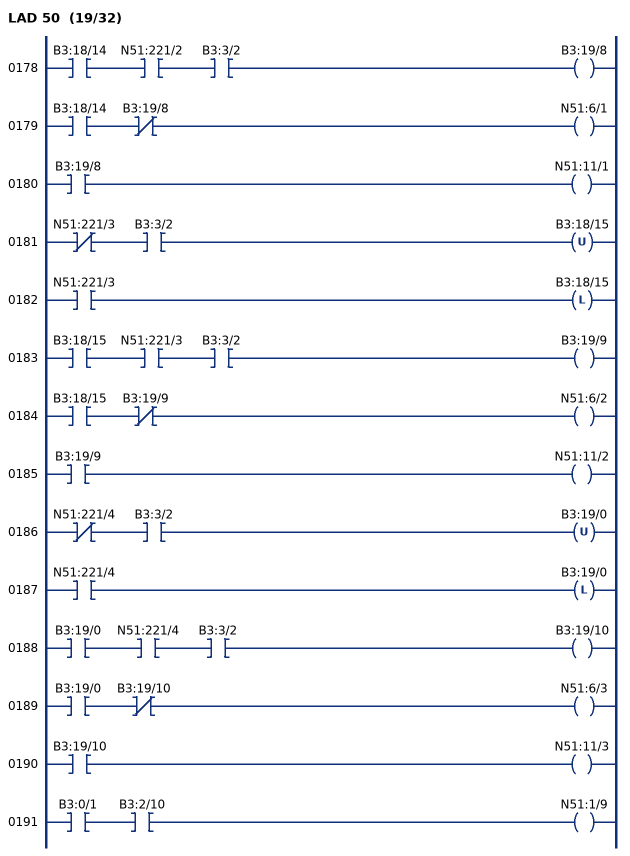
% Rung: 178 %
SOR XIC B3:18/14 XIC N51:221/2 XIC B3:3/2 OTE B3:19/8 EOR
% Rung: 179 %
SOR XIC B3:18/14 XIO B3:19/8 OTE N51:6/1 EOR
% Rung: 180 %
SOR XIC B3:19/8 OTE N51:11/1 EOR
% Rung: 181 %
SOR XIO N51:221/3 XIC B3:3/2 OTU B3:18/15 EOR
% Rung: 182 %
SOR XIC N51:221/3 OTL B3:18/15 EOR
% Rung: 183 %
SOR XIC B3:18/15 XIC N51:221/3 XIC B3:3/2 OTE B3:19/9 EOR
% Rung: 184 %
SOR XIC B3:18/15 XIO B3:19/9 OTE N51:6/2 EOR
% Rung: 185 %
SOR XIC B3:19/9 OTE N51:11/2 EOR
% Rung: 186 %
SOR XIO N51:221/4 XIC B3:3/2 OTU B3:19/0 EOR
% Rung: 187 %
SOR XIC N51:221/4 OTL B3:19/0 EOR
% Rung: 188 %
SOR XIC B3:19/0 XIC N51:221/4 XIC B3:3/2 OTE B3:19/10 EOR
% Rung: 189 %
SOR XIC B3:19/0 XIO B3:19/10 OTE N51:6/3 EOR
% Rung: 190 %
SOR XIC B3:19/10 OTE N51:11/3 EOR
% Rung: 191 %
SOR XIC B3:0/1 XIC B3:2/10 OTE N51:1/9 EOR

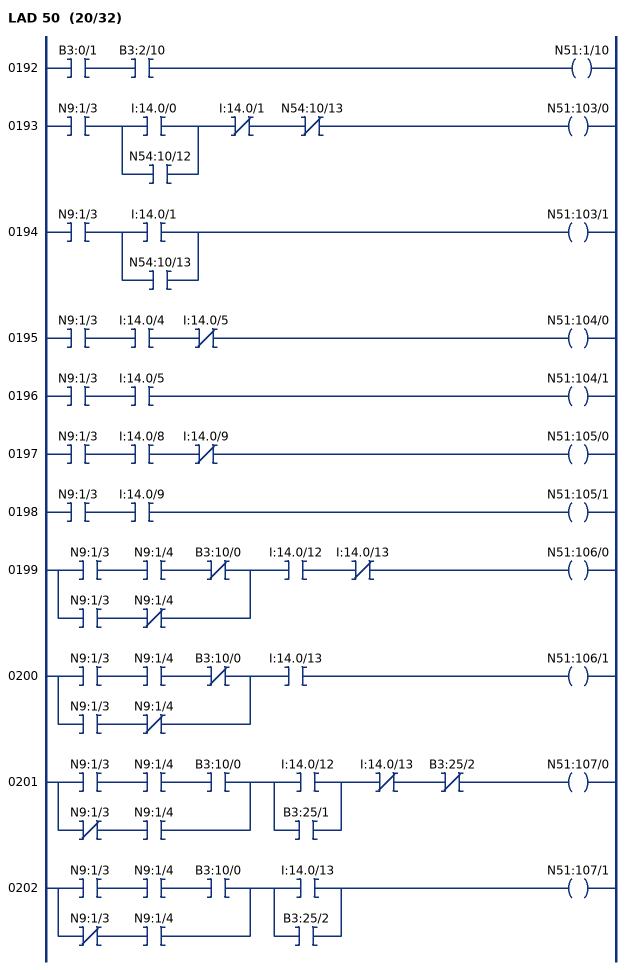
% Rung: 192 %
SOR XIC B3:0/1 XIC B3:2/10 OTE N51:1/10 EOR
% Rung: 193 %
SOR XIC N9:1/3 BST XIC I:14.0/0 NXB XIC N54:10/12 BND XIO I:14.0/1 XIO N54:10/13 OTE N51:103/0 EOR
% Rung: 194 %
SOR XIC N9:1/3 BST XIC I:14.0/1 NXB XIC N54:10/13 BND OTE N51:103/1 EOR
% Rung: 195 %
SOR XIC N9:1/3 XIC I:14.0/4 XIO I:14.0/5 OTE N51:104/0 EOR
% Rung: 196 %
SOR XIC N9:1/3 XIC I:14.0/5 OTE N51:104/1 EOR
% Rung: 197 %
SOR XIC N9:1/3 XIC I:14.0/8 XIO I:14.0/9 OTE N51:105/0 EOR
% Rung: 198 %
SOR XIC N9:1/3 XIC I:14.0/9 OTE N51:105/1 EOR
% Rung: 199 %
SOR BST XIC N9:1/3 XIC N9:1/4 XIO B3:10/0 NXB XIC N9:1/3 XIO N9:1/4 BND XIC I:14.0/12 XIO I:14.0/13 OTE N51:106/0 EOR
% Rung: 200 %
SOR BST XIC N9:1/3 XIC N9:1/4 XIO B3:10/0 NXB XIC N9:1/3 XIO N9:1/4 BND XIC I:14.0/13 OTE N51:106/1 EOR
% Rung: 201 %
SOR BST XIC N9:1/3 XIC N9:1/4 XIC B3:10/0 NXB XIO N9:1/3 XIC N9:1/4 BND BST XIC I:14.0/12 NXB XIC B3:25/1 BND XIO I:14.0/13 XIO B3:25/2 OTE N51:107/0 EOR
% Rung: 202 %
SOR BST XIC N9:1/3 XIC N9:1/4 XIC B3:10/0 NXB XIO N9:1/3 XIC N9:1/4 BND BST XIC I:14.0/13 NXB XIC B3:25/2 BND OTE N51:107/1 EOR

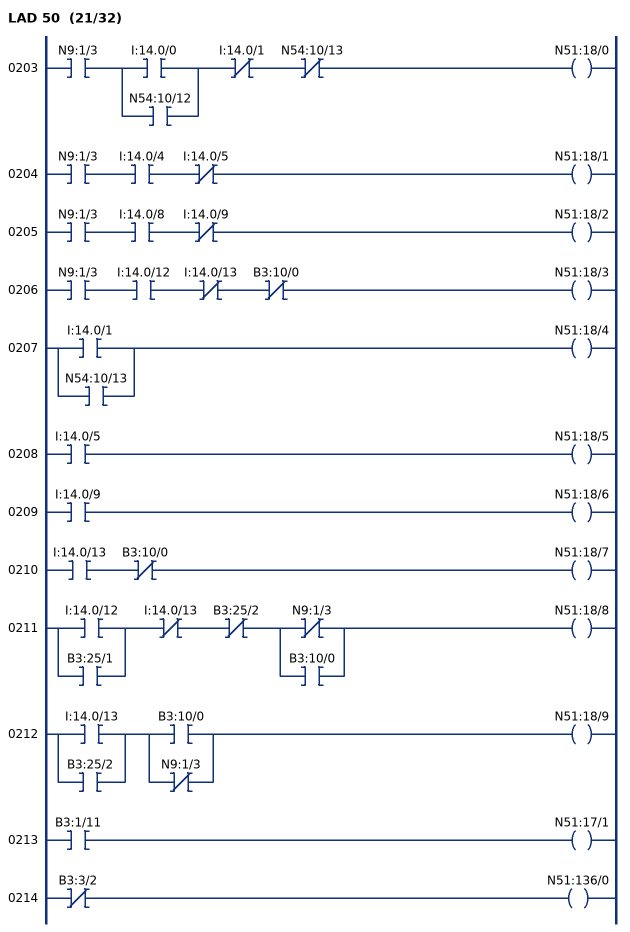
% Rung: 203 %
SOR XIC N9:1/3 BST XIC I:14.0/0 NXB XIC N54:10/12 BND XIO I:14.0/1 XIO N54:10/13 OTE N51:18/0 EOR
% Rung: 204 %
SOR XIC N9:1/3 XIC I:14.0/4 XIO I:14.0/5 OTE N51:18/1 EOR
% Rung: 205 %
SOR XIC N9:1/3 XIC I:14.0/8 XIO I:14.0/9 OTE N51:18/2 EOR
% Rung: 206 %
SOR XIC N9:1/3 XIC I:14.0/12 XIO I:14.0/13 XIO B3:10/0 OTE N51:18/3 EOR
% Rung: 207 %
SOR BST XIC I:14.0/1 NXB XIC N54:10/13 BND OTE N51:18/4 EOR
% Rung: 208 %
SOR XIC I:14.0/5 OTE N51:18/5 EOR
% Rung: 209 %
SOR XIC I:14.0/9 OTE N51:18/6 EOR
% Rung: 210 %
SOR XIC I:14.0/13 XIO B3:10/0 OTE N51:18/7 EOR
% Rung: 211 %
SOR BST XIC I:14.0/12 NXB XIC B3:25/1 BND XIO I:14.0/13 XIO B3:25/2 BST XIO N9:1/3 NXB XIC B3:10/0 BND OTE N51:18/8 EOR
% Rung: 212 %
SOR BST XIC I:14.0/13 NXB XIC B3:25/2 BND BST XIC B3:10/0 NXB XIO N9:1/3 BND OTE N51:18/9 EOR
% Rung: 213 %
SOR XIC B3:1/11 OTE N51:17/1 EOR
% Rung: 214 %
SOR XIO B3:3/2 OTE N51:136/0 EOR

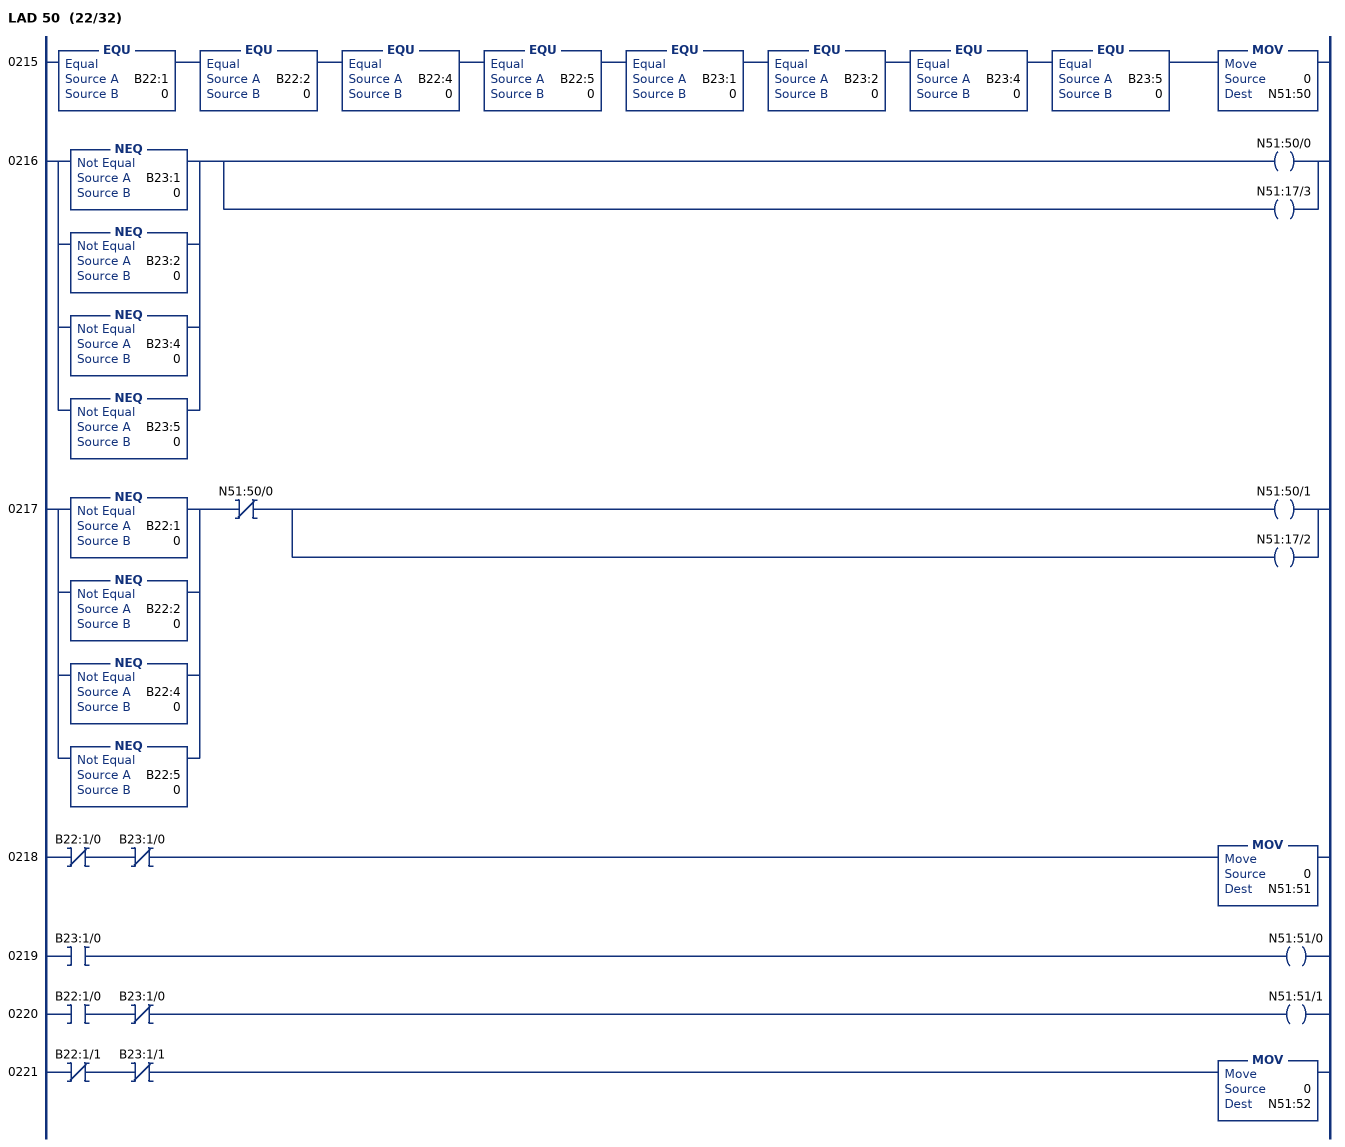
% Rung: 215 %
SOR EQU B22:1 0 EQU B22:2 0 EQU B22:4 0 EQU B22:5 0 EQU B23:1 0 EQU B23:2 0 EQU B23:4 0 EQU B23:5 0 MOV 0 N51:50 EOR
% Rung: 216 %
SOR BST NEQ B23:1 0 NXB NEQ B23:2 0 NXB NEQ B23:4 0 NXB NEQ B23:5 0 BND BST OTE N51:50/0 NXB OTE N51:17/3 BND EOR
% Rung: 217 %
SOR BST NEQ B22:1 0 NXB NEQ B22:2 0 NXB NEQ B22:4 0 NXB NEQ B22:5 0 BND XIO N51:50/0 BST OTE N51:50/1 NXB OTE N51:17/2 BND EOR
% Rung: 218 %
SOR XIO B22:1/0 XIO B23:1/0 MOV 0 N51:51 EOR
% Rung: 219 %
SOR XIC B23:1/0 OTE N51:51/0 EOR
% Rung: 220 %
SOR XIC B22:1/0 XIO B23:1/0 OTE N51:51/1 EOR
% Rung: 221 %
SOR XIO B22:1/1 XIO B23:1/1 MOV 0 N51:52 EOR

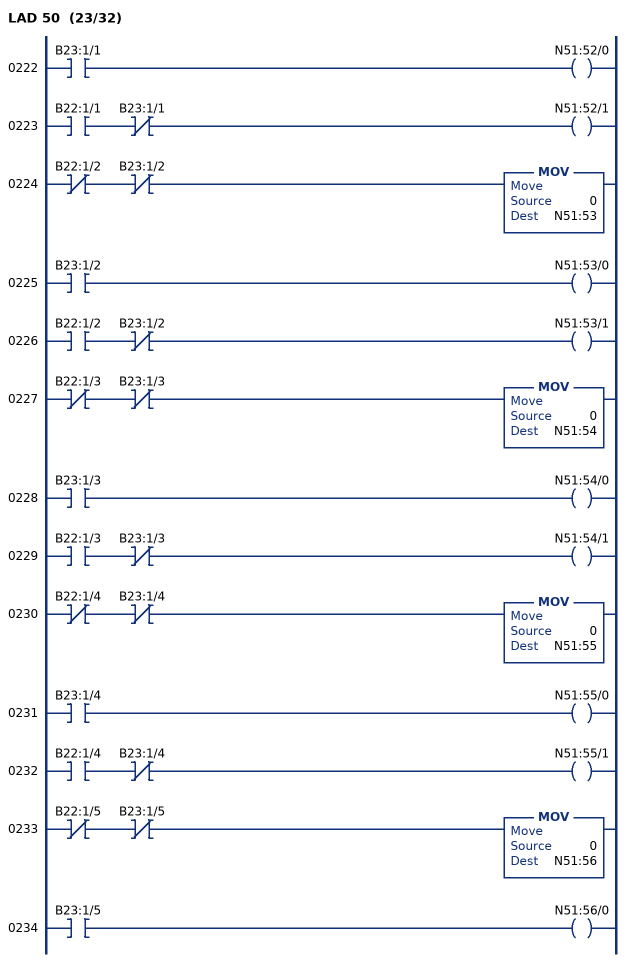
% Rung: 222 %
SOR XIC B23:1/1 OTE N51:52/0 EOR
% Rung: 223 %
SOR XIC B22:1/1 XIO B23:1/1 OTE N51:52/1 EOR
% Rung: 224 %
SOR XIO B22:1/2 XIO B23:1/2 MOV 0 N51:53 EOR
% Rung: 225 %
SOR XIC B23:1/2 OTE N51:53/0 EOR
% Rung: 226 %
SOR XIC B22:1/2 XIO B23:1/2 OTE N51:53/1 EOR
% Rung: 227 %
SOR XIO B22:1/3 XIO B23:1/3 MOV 0 N51:54 EOR
% Rung: 228 %
SOR XIC B23:1/3 OTE N51:54/0 EOR
% Rung: 229 %
SOR XIC B22:1/3 XIO B23:1/3 OTE N51:54/1 EOR
% Rung: 230 %
SOR XIO B22:1/4 XIO B23:1/4 MOV 0 N51:55 EOR
% Rung: 231 %
SOR XIC B23:1/4 OTE N51:55/0 EOR
% Rung: 232 %
SOR XIC B22:1/4 XIO B23:1/4 OTE N51:55/1 EOR
% Rung: 233 %
SOR XIO B22:1/5 XIO B23:1/5 MOV 0 N51:56 EOR
% Rung: 234 %
SOR XIC B23:1/5 OTE N51:56/0 EOR

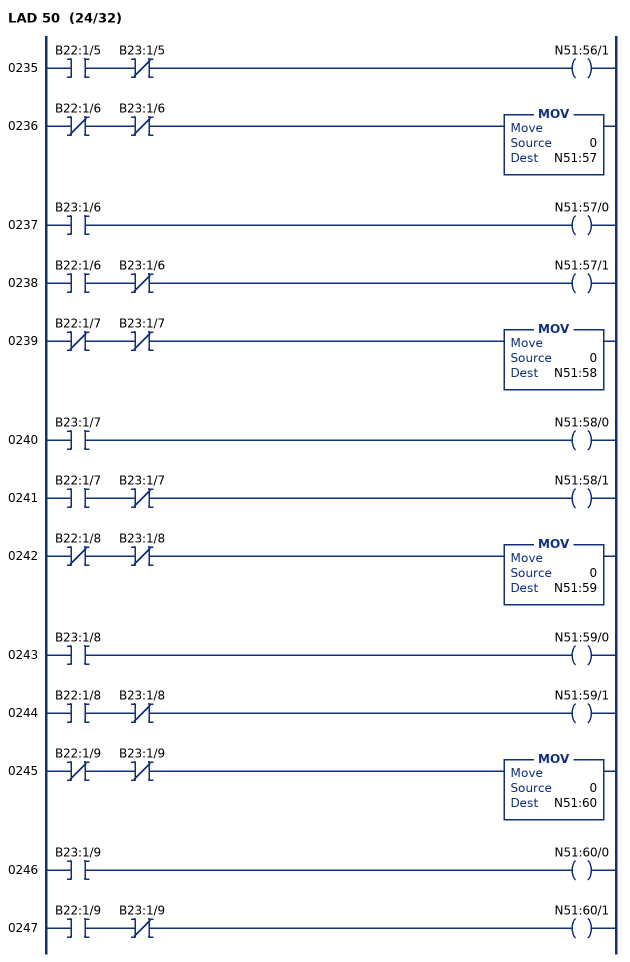
% Rung: 235 %
SOR XIC B22:1/5 XIO B23:1/5 OTE N51:56/1 EOR
% Rung: 236 %
SOR XIO B22:1/6 XIO B23:1/6 MOV 0 N51:57 EOR
% Rung: 237 %
SOR XIC B23:1/6 OTE N51:57/0 EOR
% Rung: 238 %
SOR XIC B22:1/6 XIO B23:1/6 OTE N51:57/1 EOR
% Rung: 239 %
SOR XIO B22:1/7 XIO B23:1/7 MOV 0 N51:58 EOR
% Rung: 240 %
SOR XIC B23:1/7 OTE N51:58/0 EOR
% Rung: 241 %
SOR XIC B22:1/7 XIO B23:1/7 OTE N51:58/1 EOR
% Rung: 242 %
SOR XIO B22:1/8 XIO B23:1/8 MOV 0 N51:59 EOR
% Rung: 243 %
SOR XIC B23:1/8 OTE N51:59/0 EOR
% Rung: 244 %
SOR XIC B22:1/8 XIO B23:1/8 OTE N51:59/1 EOR
% Rung: 245 %
SOR XIO B22:1/9 XIO B23:1/9 MOV 0 N51:60 EOR
% Rung: 246 %
SOR XIC B23:1/9 OTE N51:60/0 EOR
% Rung: 247 %
SOR XIC B22:1/9 XIO B23:1/9 OTE N51:60/1 EOR

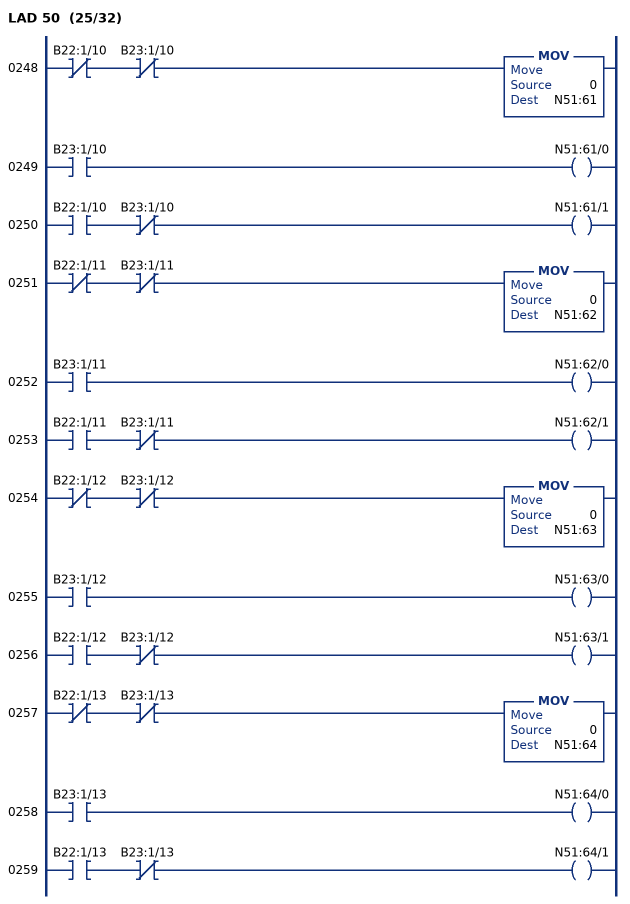
% Rung: 248 %
SOR XIO B22:1/10 XIO B23:1/10 MOV 0 N51:61 EOR
% Rung: 249 %
SOR XIC B23:1/10 OTE N51:61/0 EOR
% Rung: 250 %
SOR XIC B22:1/10 XIO B23:1/10 OTE N51:61/1 EOR
% Rung: 251 %
SOR XIO B22:1/11 XIO B23:1/11 MOV 0 N51:62 EOR
% Rung: 252 %
SOR XIC B23:1/11 OTE N51:62/0 EOR
% Rung: 253 %
SOR XIC B22:1/11 XIO B23:1/11 OTE N51:62/1 EOR
% Rung: 254 %
SOR XIO B22:1/12 XIO B23:1/12 MOV 0 N51:63 EOR
% Rung: 255 %
SOR XIC B23:1/12 OTE N51:63/0 EOR
% Rung: 256 %
SOR XIC B22:1/12 XIO B23:1/12 OTE N51:63/1 EOR
% Rung: 257 %
SOR XIO B22:1/13 XIO B23:1/13 MOV 0 N51:64 EOR
% Rung: 258 %
SOR XIC B23:1/13 OTE N51:64/0 EOR
% Rung: 259 %
SOR XIC B22:1/13 XIO B23:1/13 OTE N51:64/1 EOR

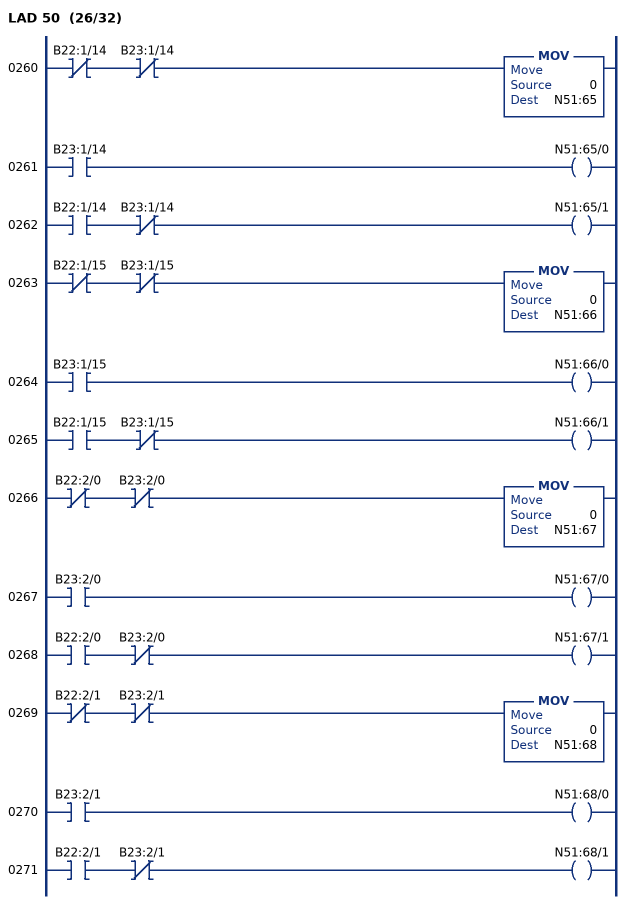
% Rung: 260 %
SOR XIO B22:1/14 XIO B23:1/14 MOV 0 N51:65 EOR
% Rung: 261 %
SOR XIC B23:1/14 OTE N51:65/0 EOR
% Rung: 262 %
SOR XIC B22:1/14 XIO B23:1/14 OTE N51:65/1 EOR
% Rung: 263 %
SOR XIO B22:1/15 XIO B23:1/15 MOV 0 N51:66 EOR
% Rung: 264 %
SOR XIC B23:1/15 OTE N51:66/0 EOR
% Rung: 265 %
SOR XIC B22:1/15 XIO B23:1/15 OTE N51:66/1 EOR
% Rung: 266 %
SOR XIO B22:2/0 XIO B23:2/0 MOV 0 N51:67 EOR
% Rung: 267 %
SOR XIC B23:2/0 OTE N51:67/0 EOR
% Rung: 268 %
SOR XIC B22:2/0 XIO B23:2/0 OTE N51:67/1 EOR
% Rung: 269 %
SOR XIO B22:2/1 XIO B23:2/1 MOV 0 N51:68 EOR
% Rung: 270 %
SOR XIC B23:2/1 OTE N51:68/0 EOR
% Rung: 271 %
SOR XIC B22:2/1 XIO B23:2/1 OTE N51:68/1 EOR

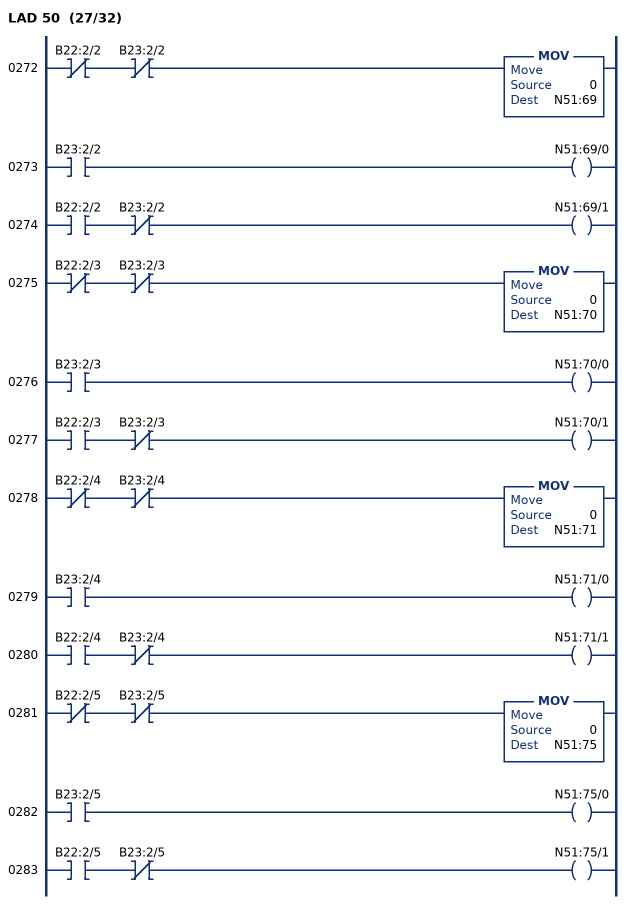
% Rung: 272 %
SOR XIO B22:2/2 XIO B23:2/2 MOV 0 N51:69 EOR
% Rung: 273 %
SOR XIC B23:2/2 OTE N51:69/0 EOR
% Rung: 274 %
SOR XIC B22:2/2 XIO B23:2/2 OTE N51:69/1 EOR
% Rung: 275 %
SOR XIO B22:2/3 XIO B23:2/3 MOV 0 N51:70 EOR
% Rung: 276 %
SOR XIC B23:2/3 OTE N51:70/0 EOR
% Rung: 277 %
SOR XIC B22:2/3 XIO B23:2/3 OTE N51:70/1 EOR
% Rung: 278 %
SOR XIO B22:2/4 XIO B23:2/4 MOV 0 N51:71 EOR
% Rung: 279 %
SOR XIC B23:2/4 OTE N51:71/0 EOR
% Rung: 280 %
SOR XIC B22:2/4 XIO B23:2/4 OTE N51:71/1 EOR
% Rung: 281 %
SOR XIO B22:2/5 XIO B23:2/5 MOV 0 N51:75 EOR
% Rung: 282 %
SOR XIC B23:2/5 OTE N51:75/0 EOR
% Rung: 283 %
SOR XIC B22:2/5 XIO B23:2/5 OTE N51:75/1 EOR

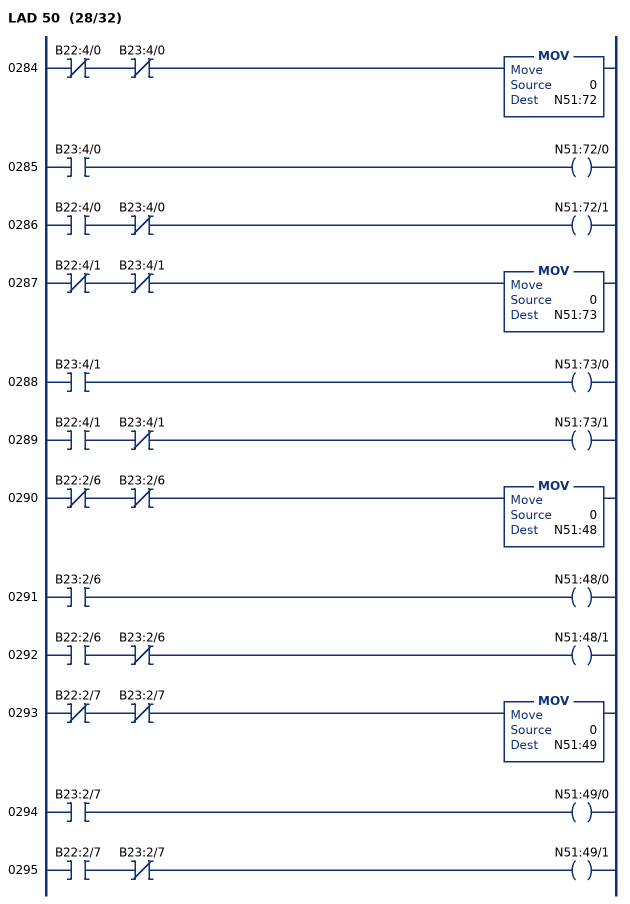
% Rung: 284 %
SOR XIO B22:4/0 XIO B23:4/0 MOV 0 N51:72 EOR
% Rung: 285 %
SOR XIC B23:4/0 OTE N51:72/0 EOR
% Rung: 286 %
SOR XIC B22:4/0 XIO B23:4/0 OTE N51:72/1 EOR
% Rung: 287 %
SOR XIO B22:4/1 XIO B23:4/1 MOV 0 N51:73 EOR
% Rung: 288 %
SOR XIC B23:4/1 OTE N51:73/0 EOR
% Rung: 289 %
SOR XIC B22:4/1 XIO B23:4/1 OTE N51:73/1 EOR
% Rung: 290 %
SOR XIO B22:2/6 XIO B23:2/6 MOV 0 N51:48 EOR
% Rung: 291 %
SOR XIC B23:2/6 OTE N51:48/0 EOR
% Rung: 292 %
SOR XIC B22:2/6 XIO B23:2/6 OTE N51:48/1 EOR
% Rung: 293 %
SOR XIO B22:2/7 XIO B23:2/7 MOV 0 N51:49 EOR
% Rung: 294 %
SOR XIC B23:2/7 OTE N51:49/0 EOR
% Rung: 295 %
SOR XIC B22:2/7 XIO B23:2/7 OTE N51:49/1 EOR

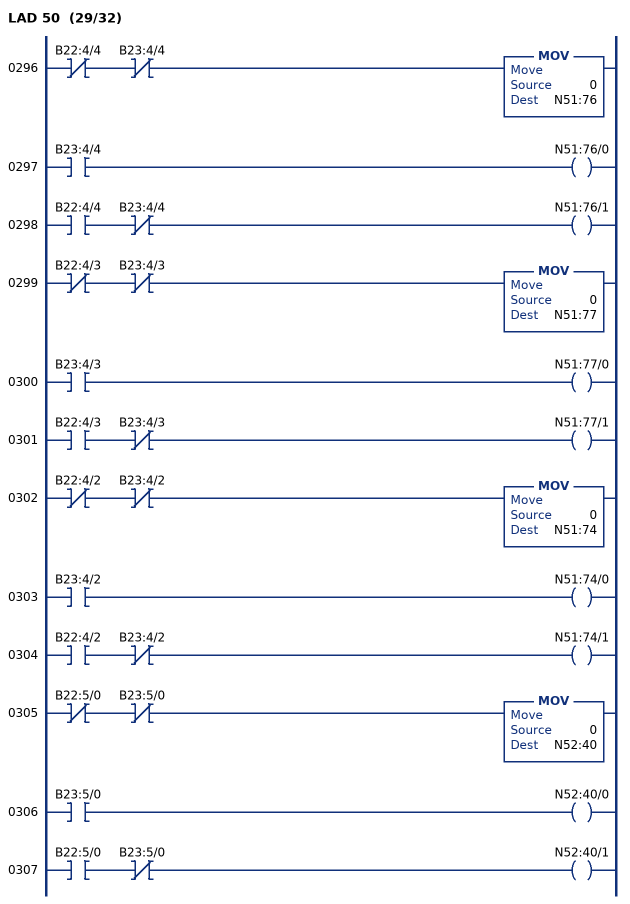
% Rung: 296 %
SOR XIO B22:4/4 XIO B23:4/4 MOV 0 N51:76 EOR
% Rung: 297 %
SOR XIC B23:4/4 OTE N51:76/0 EOR
% Rung: 298 %
SOR XIC B22:4/4 XIO B23:4/4 OTE N51:76/1 EOR
% Rung: 299 %
SOR XIO B22:4/3 XIO B23:4/3 MOV 0 N51:77 EOR
% Rung: 300 %
SOR XIC B23:4/3 OTE N51:77/0 EOR
% Rung: 301 %
SOR XIC B22:4/3 XIO B23:4/3 OTE N51:77/1 EOR
% Rung: 302 %
SOR XIO B22:4/2 XIO B23:4/2 MOV 0 N51:74 EOR
% Rung: 303 %
SOR XIC B23:4/2 OTE N51:74/0 EOR
% Rung: 304 %
SOR XIC B22:4/2 XIO B23:4/2 OTE N51:74/1 EOR
% Rung: 305 %
SOR XIO B22:5/0 XIO B23:5/0 MOV 0 N52:40 EOR
% Rung: 306 %
SOR XIC B23:5/0 OTE N52:40/0 EOR
% Rung: 307 %
SOR XIC B22:5/0 XIO B23:5/0 OTE N52:40/1 EOR

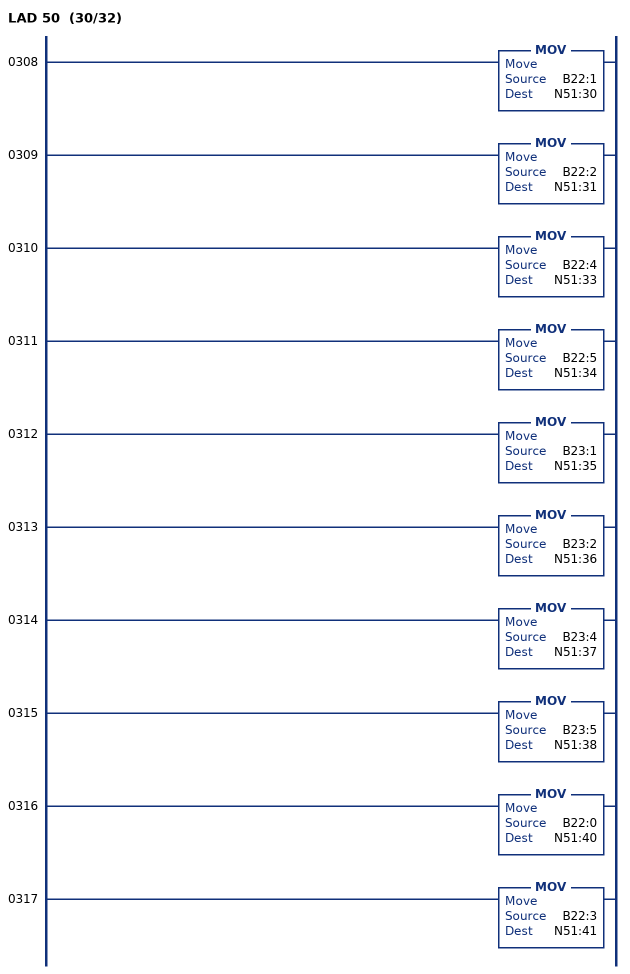
% Rung: 308 %
SOR MOV B22:1 N51:30 EOR
% Rung: 309 %
SOR MOV B22:2 N51:31 EOR
% Rung: 310 %
SOR MOV B22:4 N51:33 EOR
% Rung: 311 %
SOR MOV B22:5 N51:34 EOR
% Rung: 312 %
SOR MOV B23:1 N51:35 EOR
% Rung: 313 %
SOR MOV B23:2 N51:36 EOR
% Rung: 314 %
SOR MOV B23:4 N51:37 EOR
% Rung: 315 %
SOR MOV B23:5 N51:38 EOR
% Rung: 316 %
SOR MOV B22:0 N51:40 EOR
% Rung: 317 %
SOR MOV B22:3 N51:41 EOR

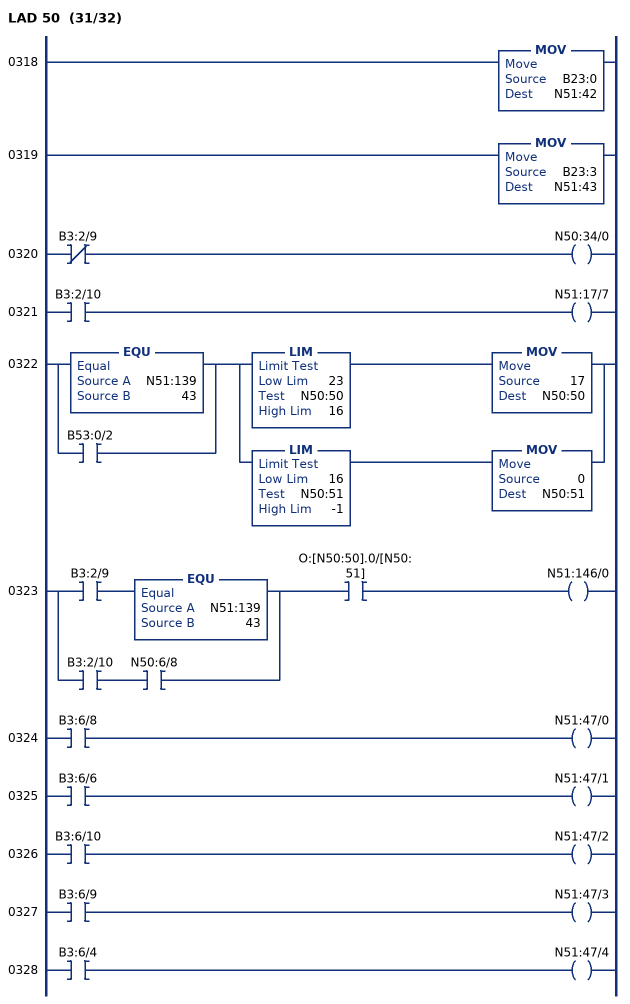
% Rung: 318 %
SOR MOV B23:0 N51:42 EOR
% Rung: 319 %
SOR MOV B23:3 N51:43 EOR
% Rung: 320 %
SOR XIO B3:2/9 OTE N50:34/0 EOR
% Rung: 321 %
SOR XIC B3:2/10 OTE N51:17/7 EOR
% Rung: 322 %
SOR BST EQU N51:139 43 NXB XIC B53:0/2 BND BST LIM 23 N50:50 16 MOV 17 N50:50 NXB LIM 16 N50:51 -1 MOV 0 N50:51 BND EOR
% Rung: 323 %
SOR BST XIC B3:2/9 EQU N51:139 43 NXB XIC B3:2/10 XIC N50:6/8 BND XIC O:[N50:50].0/[N50:51] OTE N51:146/0 EOR
% Rung: 324 %
SOR XIC B3:6/8 OTE N51:47/0 EOR
% Rung: 325 %
SOR XIC B3:6/6 OTE N51:47/1 EOR
% Rung: 326 %
SOR XIC B3:6/10 OTE N51:47/2 EOR
% Rung: 327 %
SOR XIC B3:6/9 OTE N51:47/3 EOR
% Rung: 328 %
SOR XIC B3:6/4 OTE N51:47/4 EOR

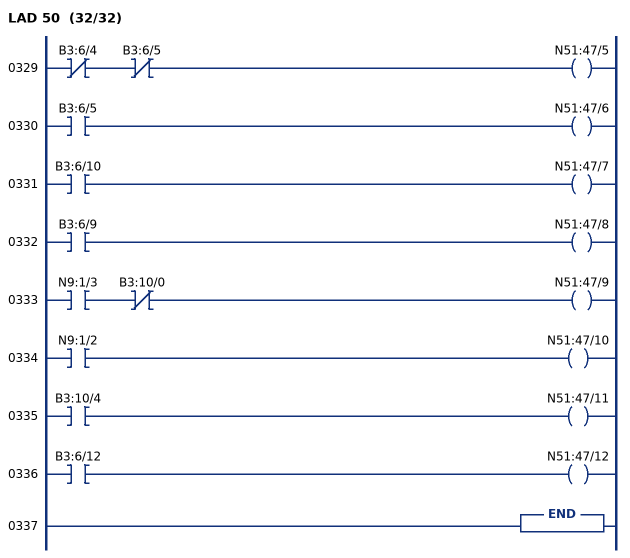
% Rung: 329 %
SOR XIO B3:6/4 XIO B3:6/5 OTE N51:47/5 EOR
% Rung: 330 %
SOR XIC B3:6/5 OTE N51:47/6 EOR
% Rung: 331 %
SOR XIC B3:6/10 OTE N51:47/7 EOR
% Rung: 332 %
SOR XIC B3:6/9 OTE N51:47/8 EOR
% Rung: 333 %
SOR XIC N9:1/3 XIO B3:10/0 OTE N51:47/9 EOR
% Rung: 334 %
SOR XIC N9:1/2 OTE N51:47/10 EOR
% Rung: 335 %
SOR XIC B3:10/4 OTE N51:47/11 EOR
% Rung: 336 %
SOR XIC B3:6/12 OTE N51:47/12 EOR
% Rung: 337 %
SOR END EOR

LADDER 51
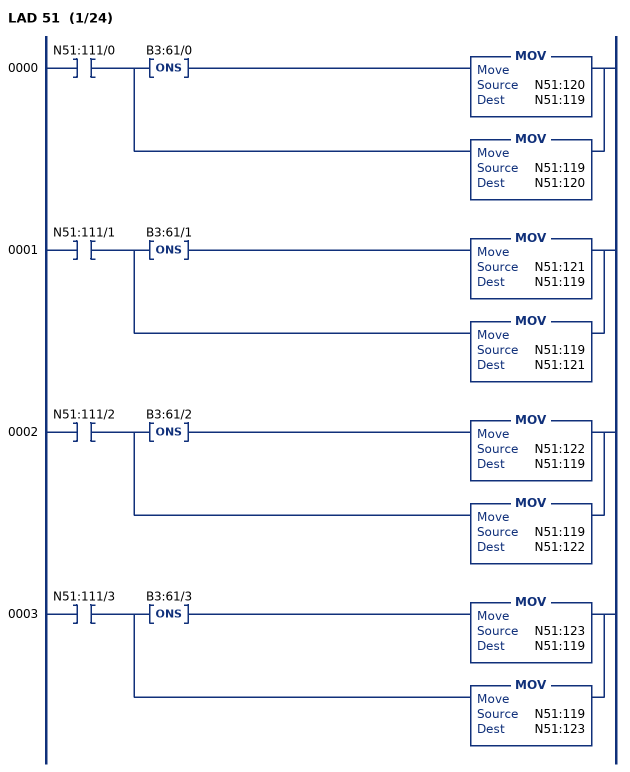
% Rung: 0 %
SOR XIC N51:111/0 BST OSR B3:61/0 MOV N51:120 N51:119 NXB MOV N51:119 N51:120 BND EOR
% Rung: 1 %
SOR XIC N51:111/1 BST OSR B3:61/1 MOV N51:121 N51:119 NXB MOV N51:119 N51:121 BND EOR
% Rung: 2 %
SOR XIC N51:111/2 BST OSR B3:61/2 MOV N51:122 N51:119 NXB MOV N51:119 N51:122 BND EOR
% Rung: 3 %
SOR XIC N51:111/3 BST OSR B3:61/3 MOV N51:123 N51:119 NXB MOV N51:119 N51:123 BND EOR

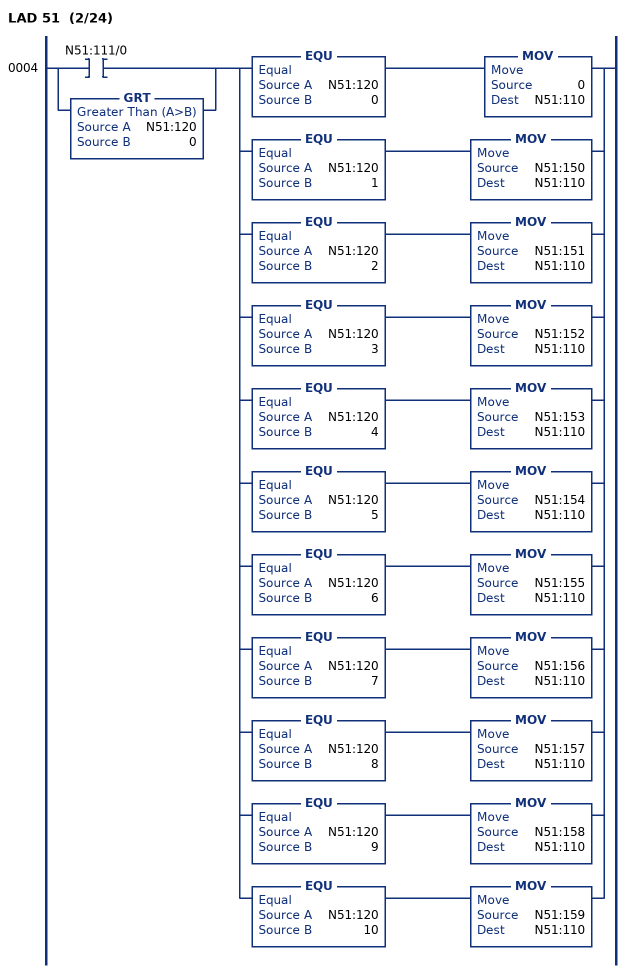
% Rung: 4 %
SOR BST XIC N51:111/0 NXB GRT N51:120 0 BND BST EQU N51:120 0 MOV 0 N51:110 NXB EQU N51:120 1 MOV N51:150 N51:110 NXB EQU N51:120 2 MOV N51:151 N51:110 NXB EQU N51:120 3 MOV N51:152 N51:110 NXB EQU N51:120 4 MOV N51:153 N51:110 NXB EQU N51:120 5 MOV N51:154 N51:110 NXB EQU N51:120 6 MOV N51:155 N51:110 NXB EQU N51:120 7 MOV N51:156 N51:110 NXB EQU N51:120 8 MOV N51:157 N51:110 NXB EQU N51:120 9 MOV N51:158 N51:110 NXB EQU N51:120 10 MOV N51:159 N51:110 BND EOR

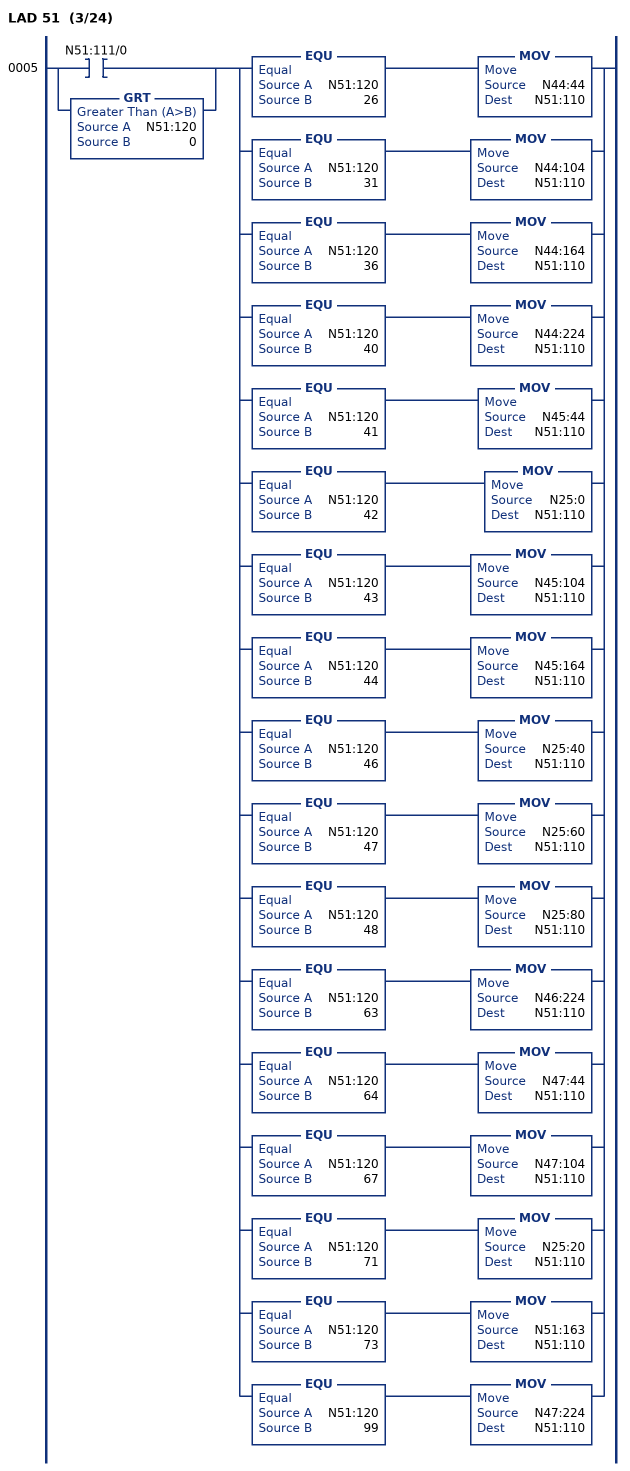
% Rung: 5 %
SOR BST XIC N51:111/0 NXB GRT N51:120 0 BND BST EQU N51:120 26 MOV N44:44 N51:110 NXB EQU N51:120 31 MOV N44:104 N51:110 NXB EQU N51:120 36 MOV N44:164 N51:110 NXB EQU N51:120 40 MOV N44:224 N51:110 NXB EQU N51:120 41 MOV N45:44 N51:110 NXB EQU N51:120 42 MOV N25:0 N51:110 NXB EQU N51:120 43 MOV N45:104 N51:110 NXB EQU N51:120 44 MOV N45:164 N51:110 NXB EQU N51:120 46 MOV N25:40 N51:110 NXB EQU N51:120 47 MOV N25:60 N51:110 NXB EQU N51:120 48 MOV N25:80 N51:110 NXB EQU N51:120 63 MOV N46:224 N51:110 NXB EQU N51:120 64 MOV N47:44 N51:110 NXB EQU N51:120 67 MOV N47:104 N51:110 NXB EQU N51:120 71 MOV N25:20 N51:110 NXB EQU N51:120 73 MOV N51:163 N51:110 NXB EQU N51:120 99 MOV N47:224 N51:110 BND EOR

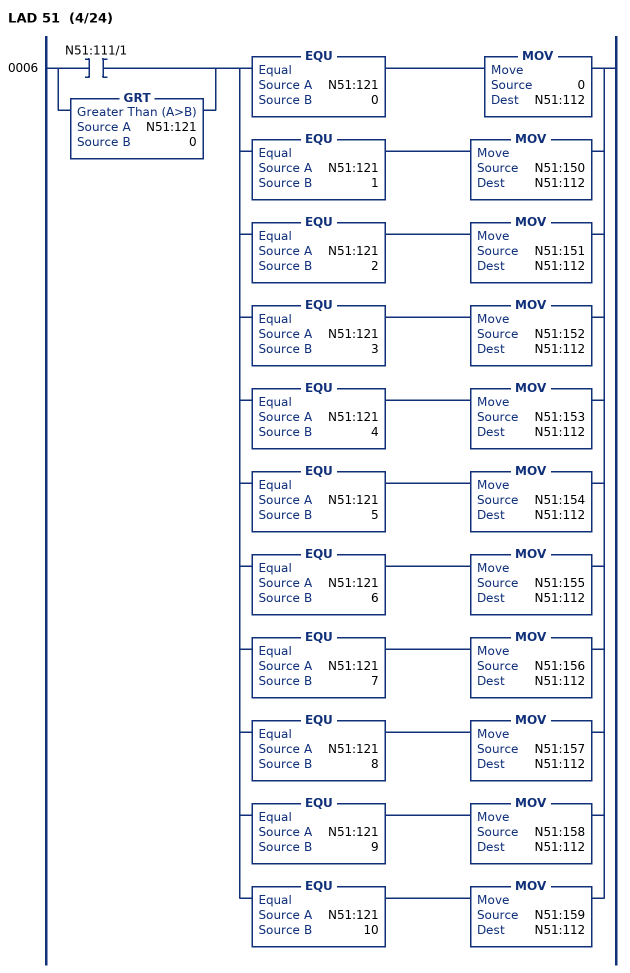
% Rung: 6 %
SOR BST XIC N51:111/1 NXB GRT N51:121 0 BND BST EQU N51:121 0 MOV 0 N51:112 NXB EQU N51:121 1 MOV N51:150 N51:112 NXB EQU N51:121 2 MOV N51:151 N51:112 NXB EQU N51:121 3 MOV N51:152 N51:112 NXB EQU N51:121 4 MOV N51:153 N51:112 NXB EQU N51:121 5 MOV N51:154 N51:112 NXB EQU N51:121 6 MOV N51:155 N51:112 NXB EQU N51:121 7 MOV N51:156 N51:112 NXB EQU N51:121 8 MOV N51:157 N51:112 NXB EQU N51:121 9 MOV N51:158 N51:112 NXB EQU N51:121 10 MOV N51:159 N51:112 BND EOR

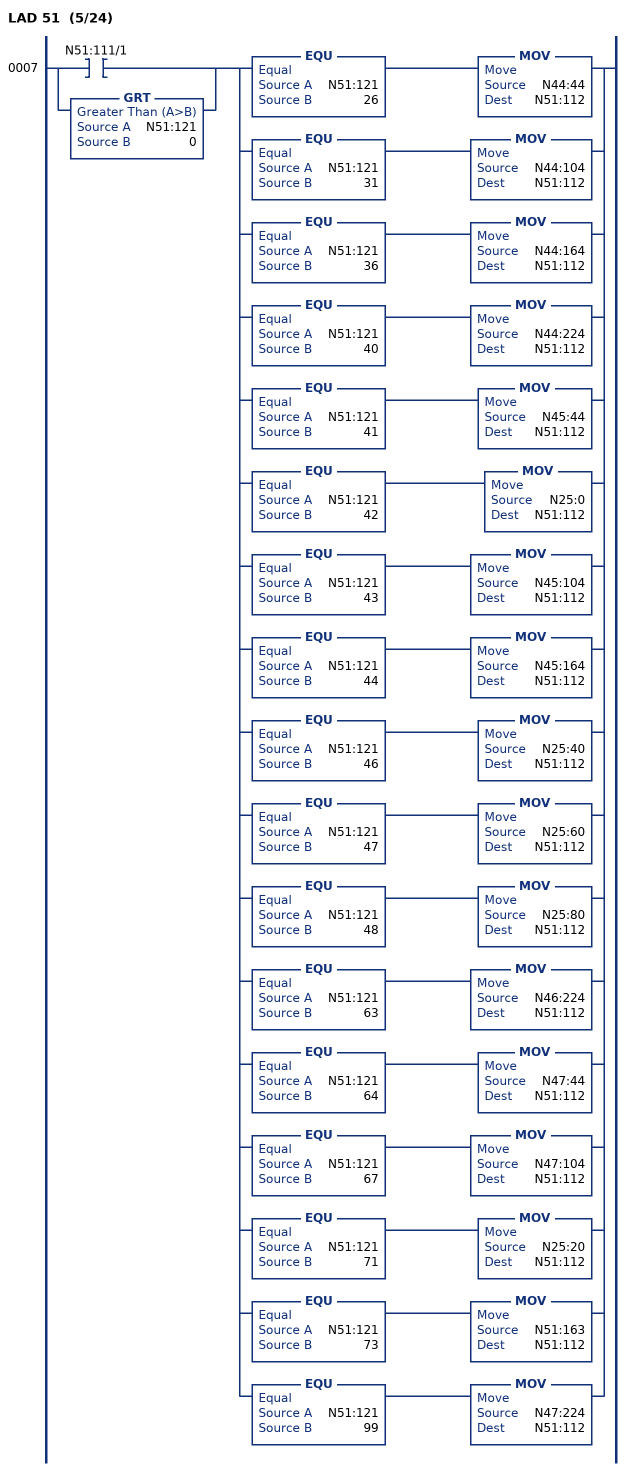
% Rung: 7 %
SOR BST XIC N51:111/1 NXB GRT N51:121 0 BND BST EQU N51:121 26 MOV N44:44 N51:112 NXB EQU N51:121 31 MOV N44:104 N51:112 NXB EQU N51:121 36 MOV N44:164 N51:112 NXB EQU N51:121 40 MOV N44:224 N51:112 NXB EQU N51:121 41 MOV N45:44 N51:112 NXB EQU N51:121 42 MOV N25:0 N51:112 NXB EQU N51:121 43 MOV N45:104 N51:112 NXB EQU N51:121 44 MOV N45:164 N51:112 NXB EQU N51:121 46 MOV N25:40 N51:112 NXB EQU N51:121 47 MOV N25:60 N51:112 NXB EQU N51:121 48 MOV N25:80 N51:112 NXB EQU N51:121 63 MOV N46:224 N51:112 NXB EQU N51:121 64 MOV N47:44 N51:112 NXB EQU N51:121 67 MOV N47:104 N51:112 NXB EQU N51:121 71 MOV N25:20 N51:112 NXB EQU N51:121 73 MOV N51:163 N51:112 NXB EQU N51:121 99 MOV N47:224 N51:112 BND EOR

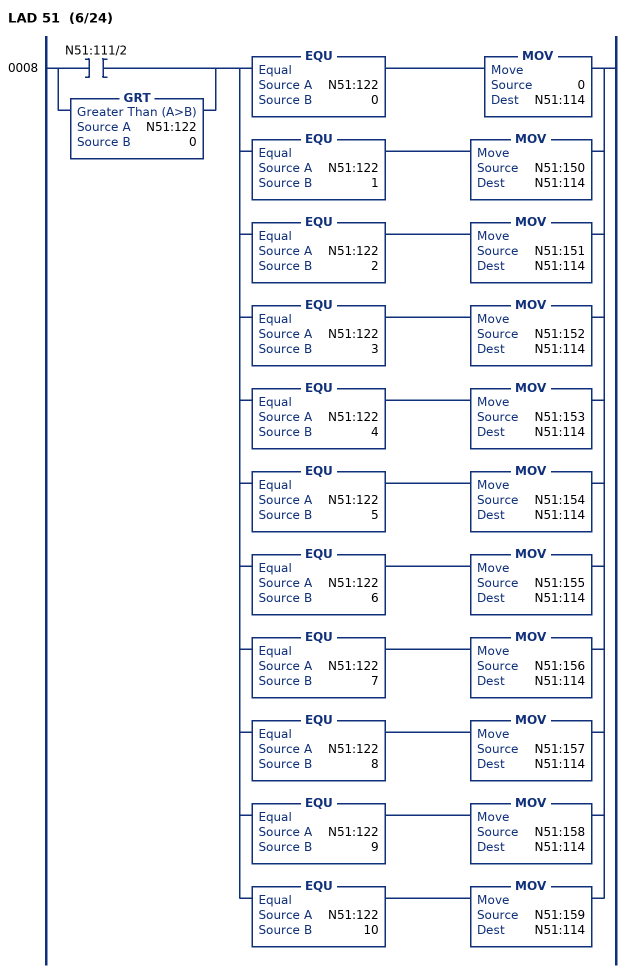
% Rung: 8 %
SOR BST XIC N51:111/2 NXB GRT N51:122 0 BND BST EQU N51:122 0 MOV 0 N51:114 NXB EQU N51:122 1 MOV N51:150 N51:114 NXB EQU N51:122 2 MOV N51:151 N51:114 NXB EQU N51:122 3 MOV N51:152 N51:114 NXB EQU N51:122 4 MOV N51:153 N51:114 NXB EQU N51:122 5 MOV N51:154 N51:114 NXB EQU N51:122 6 MOV N51:155 N51:114 NXB EQU N51:122 7 MOV N51:156 N51:114 NXB EQU N51:122 8 MOV N51:157 N51:114 NXB EQU N51:122 9 MOV N51:158 N51:114 NXB EQU N51:122 10 MOV N51:159 N51:114 BND EOR

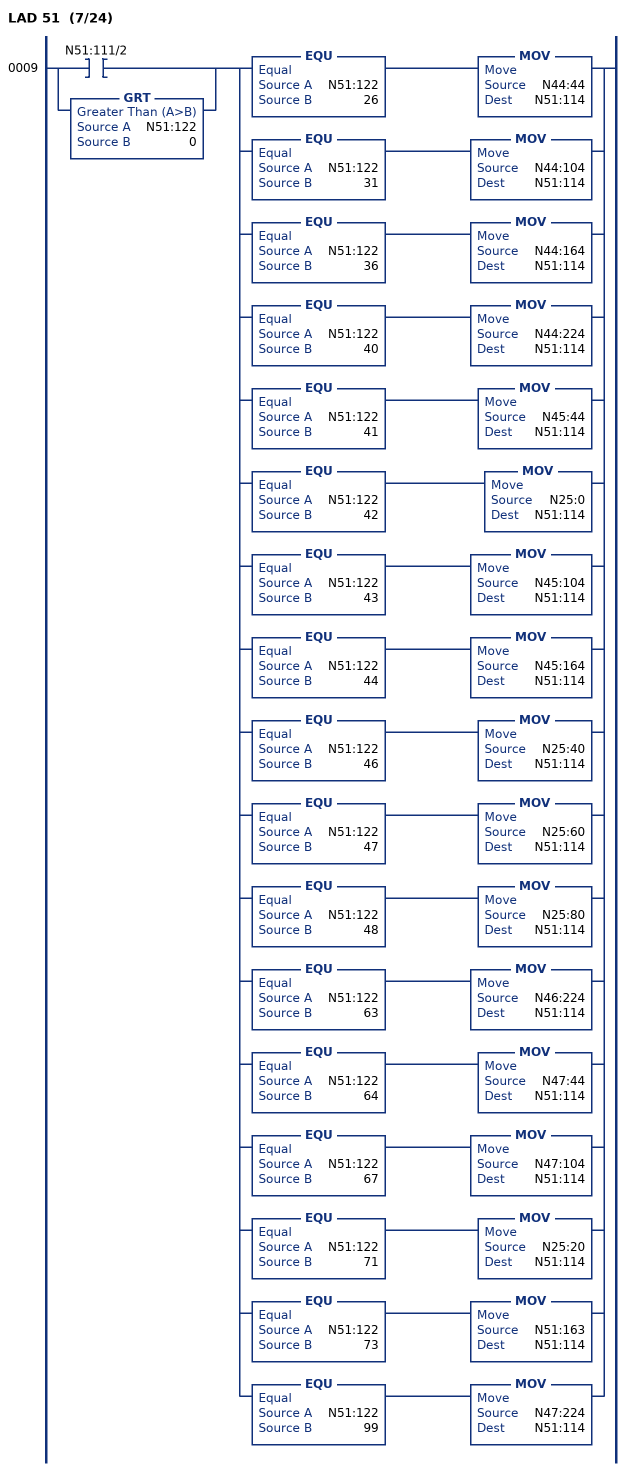
% Rung: 9 %
SOR BST XIC N51:111/2 NXB GRT N51:122 0 BND BST EQU N51:122 26 MOV N44:44 N51:114 NXB EQU N51:122 31 MOV N44:104 N51:114 NXB EQU N51:122 36 MOV N44:164 N51:114 NXB EQU N51:122 40 MOV N44:224 N51:114 NXB EQU N51:122 41 MOV N45:44 N51:114 NXB EQU N51:122 42 MOV N25:0 N51:114 NXB EQU N51:122 43 MOV N45:104 N51:114 NXB EQU N51:122 44 MOV N45:164 N51:114 NXB EQU N51:122 46 MOV N25:40 N51:114 NXB EQU N51:122 47 MOV N25:60 N51:114 NXB EQU N51:122 48 MOV N25:80 N51:114 NXB EQU N51:122 63 MOV N46:224 N51:114 NXB EQU N51:122 64 MOV N47:44 N51:114 NXB EQU N51:122 67 MOV N47:104 N51:114 NXB EQU N51:122 71 MOV N25:20 N51:114 NXB EQU N51:122 73 MOV N51:163 N51:114 NXB EQU N51:122 99 MOV N47:224 N51:114 BND EOR

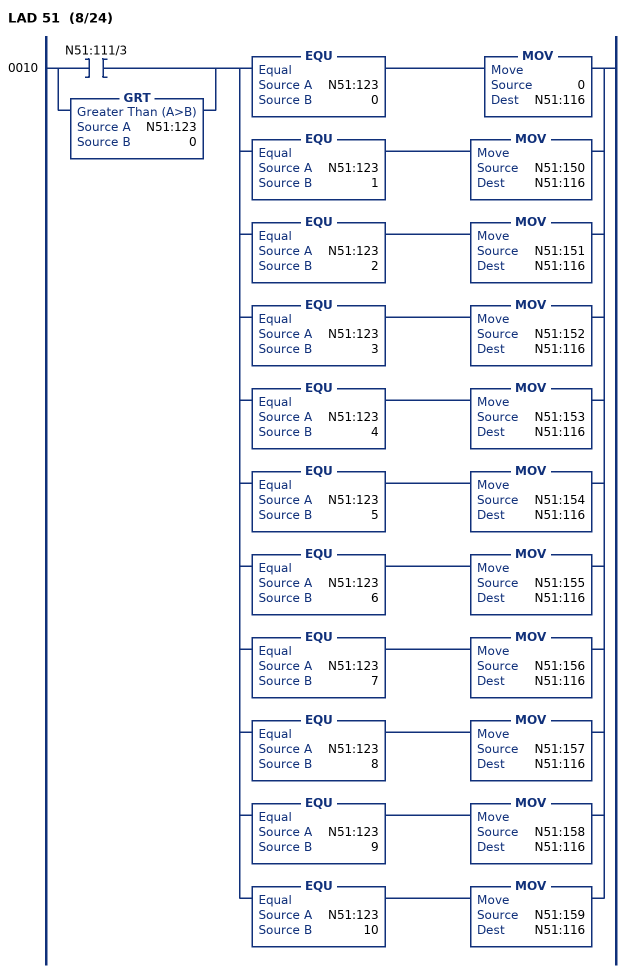
% Rung: 10 %
SOR BST XIC N51:111/3 NXB GRT N51:123 0 BND BST EQU N51:123 0 MOV 0 N51:116 NXB EQU N51:123 1 MOV N51:150 N51:116 NXB EQU N51:123 2 MOV N51:151 N51:116 NXB EQU N51:123 3 MOV N51:152 N51:116 NXB EQU N51:123 4 MOV N51:153 N51:116 NXB EQU N51:123 5 MOV N51:154 N51:116 NXB EQU N51:123 6 MOV N51:155 N51:116 NXB EQU N51:123 7 MOV N51:156 N51:116 NXB EQU N51:123 8 MOV N51:157 N51:116 NXB EQU N51:123 9 MOV N51:158 N51:116 NXB EQU N51:123 10 MOV N51:159 N51:116 BND EOR

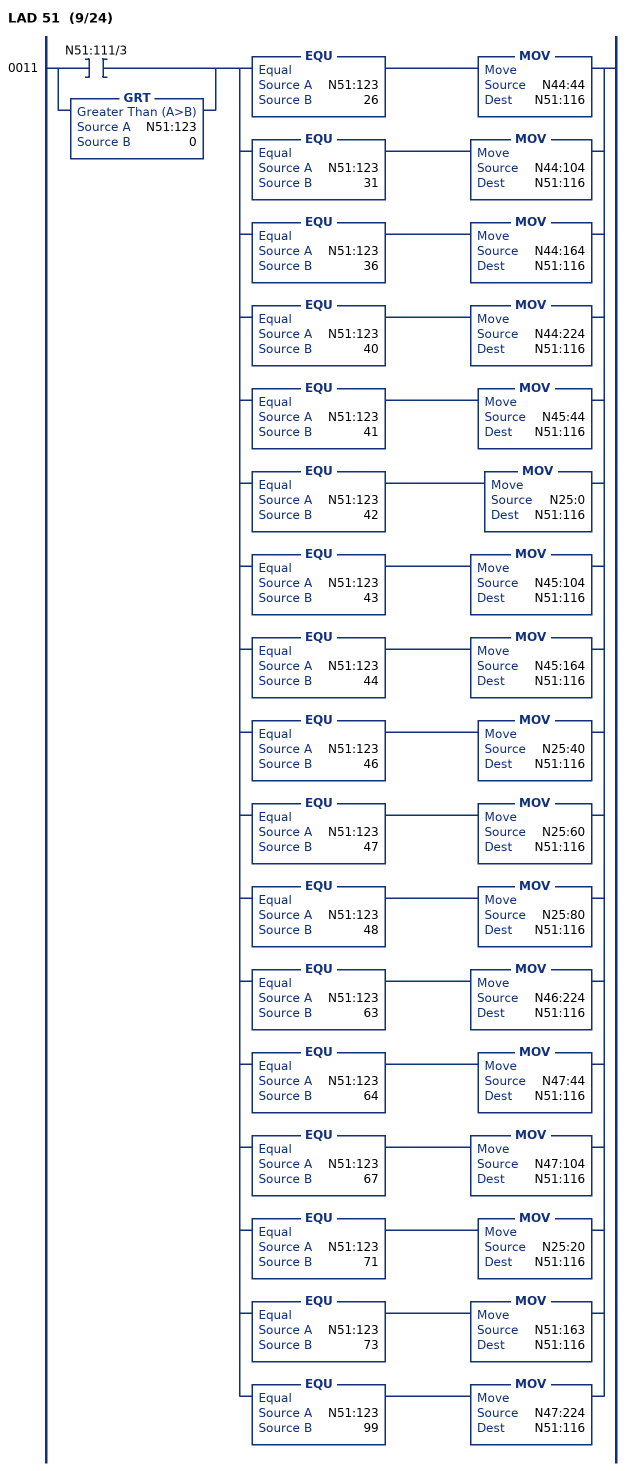
% Rung: 11 %
SOR BST XIC N51:111/3 NXB GRT N51:123 0 BND BST EQU N51:123 26 MOV N44:44 N51:116 NXB EQU N51:123 31 MOV N44:104 N51:116 NXB EQU N51:123 36 MOV N44:164 N51:116 NXB EQU N51:123 40 MOV N44:224 N51:116 NXB EQU N51:123 41 MOV N45:44 N51:116 NXB EQU N51:123 42 MOV N25:0 N51:116 NXB EQU N51:123 43 MOV N45:104 N51:116 NXB EQU N51:123 44 MOV N45:164 N51:116 NXB EQU N51:123 46 MOV N25:40 N51:116 NXB EQU N51:123 47 MOV N25:60 N51:116 NXB EQU N51:123 48 MOV N25:80 N51:116 NXB EQU N51:123 63 MOV N46:224 N51:116 NXB EQU N51:123 64 MOV N47:44 N51:116 NXB EQU N51:123 67 MOV N47:104 N51:116 NXB EQU N51:123 71 MOV N25:20 N51:116 NXB EQU N51:123 73 MOV N51:163 N51:116 NXB EQU N51:123 99 MOV N47:224 N51:116 BND EOR

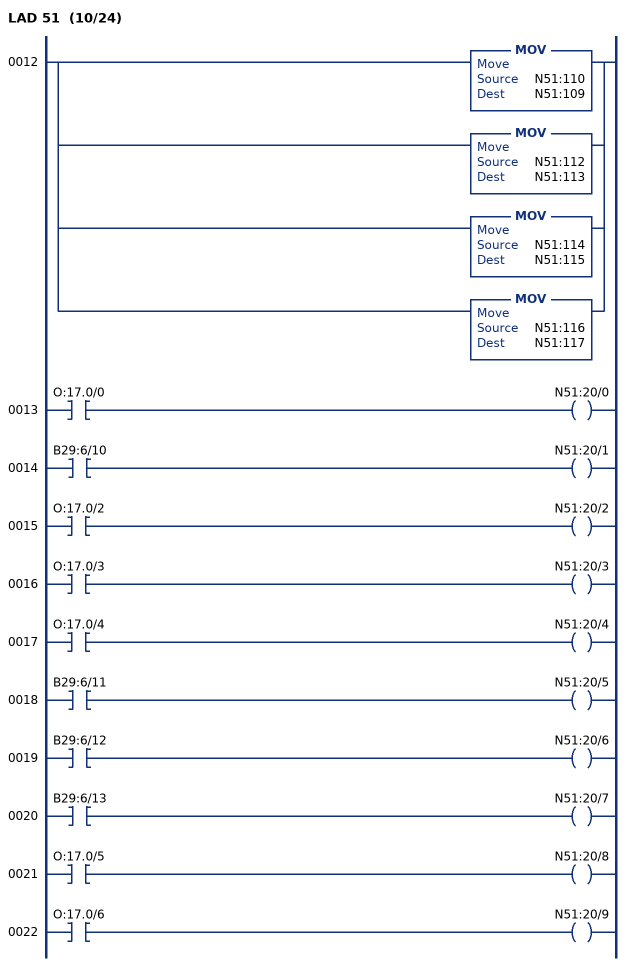
% Rung: 12 %
SOR BST MOV N51:110 N51:109 NXB MOV N51:112 N51:113 NXB MOV N51:114 N51:115 NXB MOV N51:116 N51:117 BND EOR
% Rung: 13 %
SOR XIC O:17.0/0 OTE N51:20/0 EOR
% Rung: 14 %
SOR XIC B29:6/10 OTE N51:20/1 EOR
% Rung: 15 %
SOR XIC O:17.0/2 OTE N51:20/2 EOR
% Rung: 16 %
SOR XIC O:17.0/3 OTE N51:20/3 EOR
% Rung: 17 %
SOR XIC O:17.0/4 OTE N51:20/4 EOR
% Rung: 18 %
SOR XIC B29:6/11 OTE N51:20/5 EOR
% Rung: 19 %
SOR XIC B29:6/12 OTE N51:20/6 EOR
% Rung: 20 %
SOR XIC B29:6/13 OTE N51:20/7 EOR
% Rung: 21 %
SOR XIC O:17.0/5 OTE N51:20/8 EOR
% Rung: 22 %
SOR XIC O:17.0/6 OTE N51:20/9 EOR

